PROGRAM PRG_1_PlcTask
(*
    Launch site for each component's program
    Only "fast" programs are allowed here,
    anything else needs to be relegated to a second task
*)

PRG_2_PMPS_PRE();

PRG_AT2L0_SOLID();
PRG_IM1L0_XTES();
PRG_IM1L1_PPM();
PRG_IM2L0_XTES();
PRG_IM3L0_PPM();
PRG_IM4L0_XTES();
PRG_IM5L0_PPM();
PRG_PF1L0_WFS();
PRG_RTDSL0();
PRG_SL1L0_POWER();
PRG_SL2L0_POWER();
//PRG_SP1L0_KMONO();
PRG_EM3L0_IPM();
PRG_AL1L0_REF();

PRG_3_PMPS_POST();
PRG_4_LOG();

END_PROGRAM

(* stored: Version 1.1.0.1
   POU PRG_1_PlcTask: Id {d56e695c-51d1-4f46-b1a7-5260b516ea58}, SpecialFunc None *)
